(* PLC project static_torsion.project, CODESYS CODESYS V3.5 SP17 Patch 3 *)
(* stored: creationDateTime 1970-01-01T00:00:00, modificationDateTime 2026-06-22T15:12:39.4699931 *)

PROGRAM MAIN_PRG
  VAR
    fbInit : INIT;
    lrRelativeVelocity : LREAL;  (* Параметры движения для сервопривода *)
    lrRelativeDistance : LREAL;
    lrJogVelocity : LREAL;
    xResetTorque : R_TRIG;  (* Обнуление датчиков *)
    xResetAngle : R_TRIG;
    xResetError : R_TRIG;
    xResetAlarm : R_TRIG;
    xWriteRetain : R_TRIG;  (* Запись уставок в память ПЛК *)
    wCommand : WORD;  (* Команда управления (режимы работы привода) *)
  END_VAR

            fbInit();
GVL.fbAlarm();

xResetTorque(CLK:= GVL.Control.ResetTorque);
xResetAngle(CLK:= GVL.Control.ResetAngle);
xResetError(CLK:= GVL.Control.ResetError);
xResetAlarm(CLK:= GVL.Control.ResetAlarm);
xWriteRetain(CLK:= GVL.Control.WriteRetain);

IF GVL.Control.CalibrationMode THEN
	;
END_IF

IF GVL.Control.ServiceMode THEN
	;
END_IF

IF xResetTorque.Q THEN
	GVL.iTorque_ADC_offset := GVL.iTorque_RAW;
END_IF

IF xResetAngle.Q THEN
	;
END_IF

IF xWriteRetain.Q THEN
	;
END_IF

wCommand := GetCommand(GVL.Control);

IF GVL.Control.PowerOn THEN
	GVL.fbServo.POWER_ON();
	CASE wCommand OF
		2#000:
			GVL.fbServo.HALT();
		2#001:
			GVL.fbServo.JOG_CW();
		2#010:
			GVL.fbServo.JOG_CCW();
		2#011:
			GVL.fbServo.TORQUE_HOLD();
		2#100:
			GVL.fbServo.MOVE_TO_ANGLE();
		2#101:
			;
		2#110:
			;
	END_CASE
ELSE
	GVL.fbServo.POWER_OFF();
END_IF

GVL.fbServo.RESET_ERROR(xResetError.Q);
//	GVL.fbAlarm.xAlarmReset := TRUE;

          
END_PROGRAM
